(* PLC project Generated.project, CODESYS CODESYS V3.5 SP19 Patch 1 *)
(* stored: creationDateTime 2026-08-30T22:00:23.613739, modificationDateTime 2026-08-30T22:00:23.613739 *)

(* values of E_ExtractionSequenceState: WAIT_BOTTOM_CONFIRMATION: Attente fond Kobold ou attestation opérateur; READY_TO_CLOSE: Prêt à fermer la benne; CLOSING_BUCKET: FB_Bucket ferme M2 seul; CONTROL_ASCENT: M1/M2 synchronisés au palier sans contacteur vitesse; NOMINAL_ASCENT: Montée couplée avec vitesse demandée opérateur; ERROR_HOLD: Défaut extraction, reprise interdite avant reset *)

{attribute 'qualified_only'}
{attribute 'strict'}
TYPE E_ExtractionSequenceState : (WAIT_BOTTOM_CONFIRMATION := 0, READY_TO_CLOSE := 1, CLOSING_BUCKET := 2, CONTROL_ASCENT := 3, NOMINAL_ASCENT := 4, ERROR_HOLD := 5);
END_TYPE
